// TIA Portal V17 export
// export: Created 2025-08-05T09:36:02.2665691Z, ExportSetting WithDefaults, DisplayName Totally Integrated Automation Portal, DisplayVersion V17, DisplayName TIA Portal Openness, DisplayVersion V17, DisplayName TIA Portal Version Control Interface, DisplayVersion V17, DisplayName SINAMICS Startdrive Advanced, DisplayVersion V17, DisplayName SINAMICS Startdrive G130, G150, S120, S150, SINAMICS MV, S210, DisplayVersion V17, DisplayName SINAMICS Startdrive G110M, G120, G120C, G120D, G120P, G115D, DisplayVersion V17, DisplayName STEP 7 Professional, DisplayVersion V17, DisplayName STEP 7 Safety, DisplayVersion V17, DisplayName WinCC Advanced, DisplayVersion V17
TYPE "typeSmcChillerHrle90a40cmStatus"
// stored: IsFailsafeCompliant false
   STRUCT
      fluidActualDischargeTempCh1 { ExternalAccessible := 'False'; ExternalVisible := 'False'; ExternalWritable := 'False'} : Real;   // Temperatur am Ausgang Kanal 1 / Temperature at the outlet channel 1
      fluidActualDischargeTempCh2 { ExternalAccessible := 'False'; ExternalVisible := 'False'; ExternalWritable := 'False'} : Real;   // Temperatur am Ausgang Kanal 2 / Temperature at the outlet channel 2
      fluidActualDischargePressureCh1 { ExternalAccessible := 'False'; ExternalVisible := 'False'; ExternalWritable := 'False'} : Real;   // Druck am Ausgang Kanal 1 / Pressure at the outlet channel 1
      fluidSetpointDischargeTempCh1 { ExternalAccessible := 'False'; ExternalVisible := 'False'; ExternalWritable := 'False'} : Real;   // Sollwert für die Flüssigkeitstemperatur Kanal 1 / Target value for the fluid temperature channel 1
      chillerRunning { ExternalAccessible := 'False'; ExternalVisible := 'False'; ExternalWritable := 'False'} : Bool;   // Kühlung läuft / Cooling running
      chillerInRemoteMode { ExternalAccessible := 'False'; ExternalVisible := 'False'; ExternalWritable := 'False'} : Bool;   // Kältemaschine im Remote-Modus / Cooling unit in Remote mode
      chillerTempReady { ExternalAccessible := 'False'; ExternalVisible := 'False'; ExternalWritable := 'False'} : Bool;   // Chiller-Prozessvorbereitung abgeschlossen / Chiller process preparation finished
      dataDisplay { ExternalAccessible := 'False'; ExternalVisible := 'False'; ExternalWritable := 'False'} : Struct   // Über die Datenanzeigeanweisung zurückgegebener Wert / Value returned via the data display instruction
         "1" { ExternalAccessible := 'False'; ExternalVisible := 'False'; ExternalWritable := 'False'} : Struct   // 1
            valueType { ExternalAccessible := 'False'; ExternalVisible := 'False'; ExternalWritable := 'False'} : Byte;   // Art des Wertes / Type of value
            value { ExternalAccessible := 'False'; ExternalVisible := 'False'; ExternalWritable := 'False'} : Real;   // Wert / Value
         END_STRUCT;
         "2" { ExternalAccessible := 'False'; ExternalVisible := 'False'; ExternalWritable := 'False'} : Struct   // 2
            valueType { ExternalAccessible := 'False'; ExternalVisible := 'False'; ExternalWritable := 'False'} : Byte;   // Art des Wertes / Type of value
            value { ExternalAccessible := 'False'; ExternalVisible := 'False'; ExternalWritable := 'False'} : Real;   // Wert / Value
         END_STRUCT;
      END_STRUCT;
      errorFB { ExternalAccessible := 'False'; ExternalVisible := 'False'; ExternalWritable := 'False'} : Struct   // Fehler im Funktionsblock / Error in the function block
         active { ExternalAccessible := 'False'; ExternalVisible := 'False'; ExternalWritable := 'False'} : Bool;   // Aktiv / Active
         errorLocation { ExternalAccessible := 'False'; ExternalVisible := 'False'; ExternalWritable := 'False'} : DWord;   // Ort des Fehlers / Error location
         errorCode { ExternalAccessible := 'False'; ExternalVisible := 'False'; ExternalWritable := 'False'} : DWord;   // Fehlercode / Error code
      END_STRUCT;
      alarmDevice { ExternalAccessible := 'False'; ExternalVisible := 'False'; ExternalWritable := 'False'} : Struct   // Alarm am Kühlgerät / Alarm at cooler
         active { ExternalAccessible := 'False'; ExternalVisible := 'False'; ExternalWritable := 'False'} : Bool;   // Aktiv / Active
      END_STRUCT;
      warningDevice { ExternalAccessible := 'False'; ExternalVisible := 'False'; ExternalWritable := 'False'} : Struct   // Warnung am Kühlgerät / Warning on the cooling unit
         active { ExternalAccessible := 'False'; ExternalVisible := 'False'; ExternalWritable := 'False'} : Bool;   // Aktiv / Active
      END_STRUCT;
   END_STRUCT;
END_TYPE
